FUNCTION_BLOCK ErrorCollection implements I_ErrorCollection
VAR
	errors : Stack;
END_VAR

METHOD PUBLIC GetEnumerator : I_ForwardEnumerator
VAR_INPUT
END_VAR
GetEnumerator := errors.GetEnumerator();
END_METHOD

METHOD PUBLIC Insert
VAR_INPUT
	error : I_Error;
END_VAR
errors.Push(error);
END_METHOD

END_FUNCTION_BLOCK

(* stored: Version 1.1.0.1, ProductVersion 3.1.4024.12
   POU ErrorCollection: Id {68f90357-7237-0af2-388f-e56794399946}, SpecialFunc None
   Method GetEnumerator: Id {f628d4ae-9a9e-04e7-1fb4-f954de25a9aa}
   Method Insert: Id {7e5598c6-1f95-0eb6-0614-4bf48418e5c0} *)
